// TIA Portal V20 export
TYPE "LER_typeAxisInterlockSource"
// stored: Access Published
   STRUCT
      moveVelocity : Bool;
      stop : Bool;
      fastStop : Bool;
      torqueLimiting : Bool;
      homing : Bool;
      posRelative : Bool;
      posAbsolute : Array[0..15] of Bool;
      gearInRelative : Bool;
      gearInAbsolute : Bool;
      gearInVelocity : Bool;
      camIn : Bool;
      gearOutCamOut : Bool;
      phasing : Bool;
      offset : Bool;
   END_STRUCT;
END_TYPE
